% RSLogix 500 project LVD190424_LVD.RSS, saved by version 11.00.00.00 %
PROJECT "LINCEBOT"    % processor: MicroLogix 1400 %

PROGRAM FILES
  LAD 2 "MAIN"  65 rungs  % Main Program Routine %
  LAD 4 "PACKAGER"  20 rungs  % normal %
  LAD 6 "TIMING"  11 rungs  % normal %
  LAD 8 "LOOP TIME"  6 rungs
  LAD 10 "AIR PRESUR"  2 rungs
  LAD 12 "ENABLES"  14 rungs
  LAD 14 "SPEED OUT"  12 rungs
  LAD 16 "TOTALCOUNT"  4 rungs
  LAD 18 "TESTTRIG1"  3 rungs
  LAD 20 "TESTTRIG5"  3 rungs
  LAD 22 "TESTTRIG6"  3 rungs
  LAD 24 "SKIPPED"  5 rungs
  LAD 26 "TEST TIME"  11 rungs
  LAD 70 "ALIGNFAILS"  4 rungs  % normal %
  LAD 80 "HSC BOT"  5 rungs
  LAD 90 "HSC TOP"  5 rungs
  LAD 100 "1 MS STI"  24 rungs  % high speed %
  LAD 102 "SPEED BOT"  8 rungs  % high speed %
  LAD 103 "SPEED TOP"  8 rungs  % high speed %
  LAD 104 "P BOT"  9 rungs  % high speed %
  LAD 105 "P TOP"  8 rungs  % high speed %
  LAD 110 "SHIFT BOT"  9 rungs
  LAD 111 "SHIFT TOP"  13 rungs
  LAD 120 "BOTOPTIC"  3 rungs
  LAD 121 "BOTOPTMES"  7 rungs
  LAD 124 "INS1RESULT"  10 rungs
  LAD 125 "FIXERR1"  8 rungs
  LAD 127 "INS1"  40 rungs
  LAD 128 "INS1PASS"  4 rungs
  LAD 129 "INS1ACQ"  11 rungs
  LAD 130 "INS1TRIG"  9 rungs
  LAD 131 "XFER"  2 rungs
  LAD 140 "TOPOPTIC"  7 rungs
  LAD 141 "TOPOPVERT"  3 rungs
  LAD 142 "TOPOPREAL"  7 rungs
  LAD 143 "TOPOPTEST"  15 rungs
  LAD 144 "TOPOPOKAY"  6 rungs
  LAD 149 "INS5RESULT"  10 rungs
  LAD 150 "FIXERR5"  8 rungs
  LAD 152 "INS5"  35 rungs
  LAD 153 "INS5PASS"  4 rungs
  LAD 154 "INS5ACQ"  11 rungs
  LAD 155 "INS5TRIG"  9 rungs
  LAD 159 "INS6RESULT"  10 rungs
  LAD 160 "FIXERR6"  8 rungs
  LAD 162 "INS6"  29 rungs
  LAD 163 "INS6PASS"  4 rungs
  LAD 164 "INS6ACQ"  10 rungs
  LAD 165 "INS6TRIG"  9 rungs
  LAD 170 "PASS BLOW"  11 rungs
  LAD 180 "RATE"  14 rungs
  LAD 200 "TESTOPTIC"  6 rungs
  LAD 201 "UNUSED"  19 rungs
  LAD 255 "BLANK"  11 rungs

DATA FILES
  O0 OUTPUT  11 elements
  I1 INPUT  11 elements
  S2 STATUS  66 elements
  B3 BINARY  14 elements
  T4 TIMER  40 elements
  C5 COUNTER  1 elements
  R6 CONTROL  20 elements
  N7 INTEGER  200 elements
  F8 FLOAT  100 elements
  B9 TOP BS DAT  256 elements
  B10 OLD_COM  1 elements
  B11 BOT BS DAT  256 elements
  B12 HMI_BINARY  22 elements  % general use with hmi to avoid additional reads %
  L13  COUNTS  256 elements
  F14 HMI_FLOATS  100 elements
  N15 HMI_INTS  100 elements
  L16 HMI_LONGS  100 elements
  B17 SIDE DATA  128 elements
  B18 TOP DATA  128 elements
  L19 INS1TIME  10 elements
  L20 INS1POS  10 elements
  L21 INS5TIME  10 elements
  L22 INS5POS  10 elements
  L23 NEW READ  100 elements
  L24 NEW WRITE  100 elements
  L25 INS6TIME  10 elements
  L26 INS6POS  10 elements
  L42   52 elements
  B181 BLANK  256 elements  % used to wipe bs files %
  F182 TEST FLOAT  50 elements
  L183 TEST LONG  50 elements
  N184 TEST INTS  50 elements
  B185 TEST BITS  50 elements
  N186 HMI INTS  50 elements
  L187 HMI LONG  50 elements
  F188 HMI FLOAT  50 elements
  B189 HMI BITS  50 elements
  L190 COUNTS  50 elements
  B191 ERROR BITS  10 elements
  L192 SPD OFFSET  50 elements
  F193 SPD OFFSET  50 elements
  B194 BOT GOOD  128 elements
  B195 TOP GOOD  128 elements
  B196 CTRL BITS  50 elements
  N197 CTRL INTS  50 elements
  B198 TRK BITS  50 elements
  L199 TRK LONG  50 elements
  N200 TRK INTS  50 elements
  L201 INS LONG  50 elements
  B202 INS BITS  50 elements
  N203 INS INTS  50 elements
  L204 CTRL LONG  50 elements
  F205 CTRL FLTS  50 elements

LADDER 2 "MAIN"    % Main Program Routine %
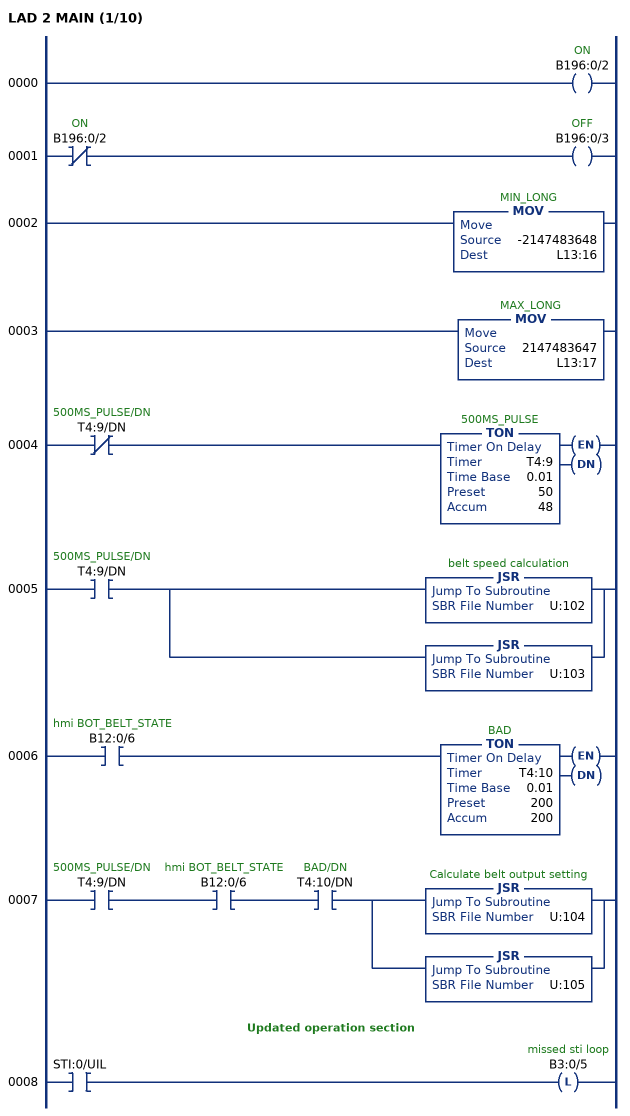
% Rung: 0 %
SOR OTE B196:0/2 EOR
%   B196:0/2  ON %
% Rung: 1 %
SOR XIO B196:0/2 OTE B196:0/3 EOR
%   B196:0/2  ON %
%   B196:0/3  OFF %
% Rung: 2 %
SOR MOV -2147483648 L13:16 EOR
%   L13:16  MIN_LONG %
% Rung: 3 %
SOR MOV 2147483647 L13:17 EOR
%   L13:17  MAX_LONG %
% Rung: 4 %
SOR XIO T4:9/DN TON T4:9 0.01 50 48 EOR
%   T4:9  500MS_PULSE %
% Rung: 5 %
SOR XIC T4:9/DN BST JSR U:102 NXB JSR U:103 BND EOR
%   T4:9  500MS_PULSE %
%   U:102  "belt speed calculation" %
% Rung: 6 %
SOR XIC B12:0/6 TON T4:10 0.01 200 200 EOR
%   B12:0/6  BOT_BELT_STATE  "hmi" %
%   T4:10  BAD %
% Rung: 7 %
SOR XIC T4:9/DN XIC B12:0/6 XIC T4:10/DN BST JSR U:104 NXB JSR U:105 BND EOR
%   T4:9  500MS_PULSE %
%   B12:0/6  BOT_BELT_STATE  "hmi" %
%   T4:10  BAD %
%   U:104  "Calculate belt output setting" %
% Rung: 8 %
% TITLE: Updated operation section %
SOR XIC STI:0/UIL OTL B3:0/5 EOR
%   B3:0/5  "missed sti loop" %

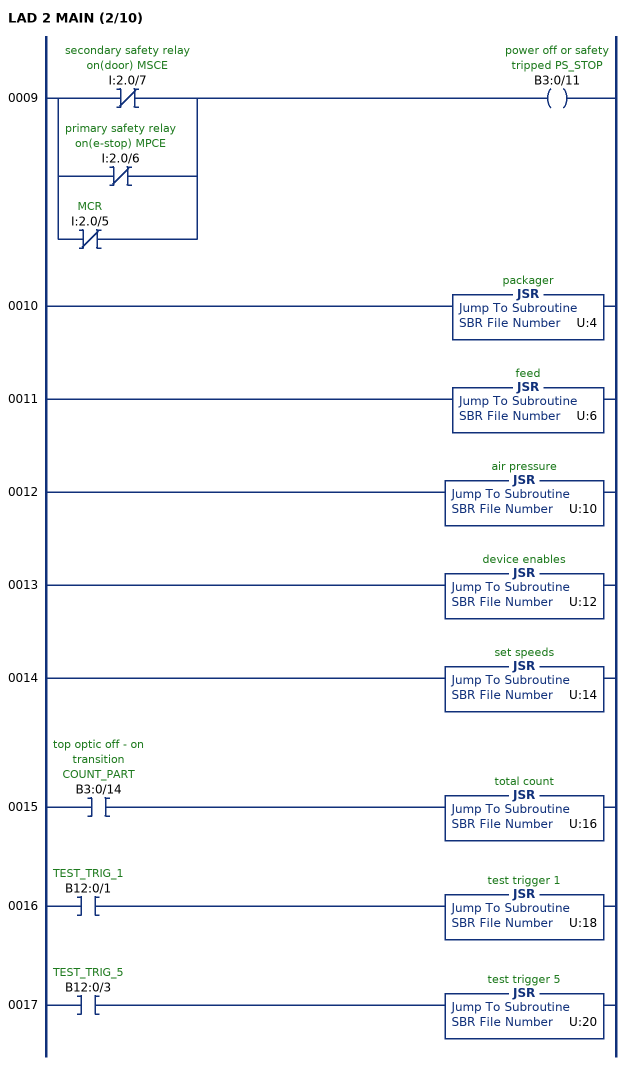
% Rung: 9 %
SOR BST XIO I:2.0/7 NXB XIO I:2.0/6 NXB XIO I:2.0/5 BND OTE B3:0/11 EOR
%   I:2.0/7  MSCE  "secondary safety relay on(door)" %
%   I:2.0/6  MPCE  "primary safety relay on(e-stop)" %
%   I:2.0/5  MCR %
%   B3:0/11  PS_STOP  "power off or safety tripped" %
% Rung: 10 %
SOR JSR U:4 EOR
%   U:4  "packager" %
% Rung: 11 %
SOR JSR U:6 EOR
%   U:6  "feed" %
% Rung: 12 %
SOR JSR U:10 EOR
%   U:10  "air pressure" %
% Rung: 13 %
SOR JSR U:12 EOR
%   U:12  "device enables" %
% Rung: 14 %
SOR JSR U:14 EOR
%   U:14  "set speeds" %
% Rung: 15 %
SOR XIC B3:0/14 JSR U:16 EOR
%   B3:0/14  COUNT_PART  "top optic off - on transition" %
%   U:16  "total count" %
% Rung: 16 %
SOR XIC B12:0/1 JSR U:18 EOR
%   B12:0/1  TEST_TRIG_1 %
%   U:18  "test trigger 1" %
% Rung: 17 %
SOR XIC B12:0/3 JSR U:20 EOR
%   B12:0/3  TEST_TRIG_5 %
%   U:20  "test trigger 5" %

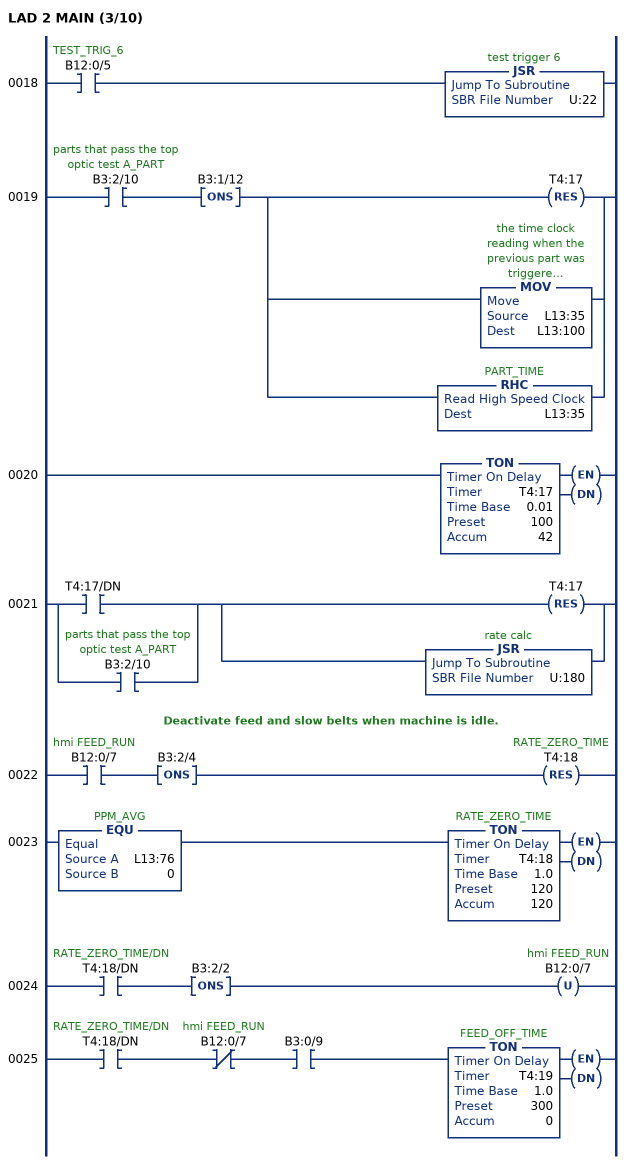
% Rung: 18 %
SOR XIC B12:0/5 JSR U:22 EOR
%   B12:0/5  TEST_TRIG_6 %
%   U:22  "test trigger 6" %
% Rung: 19 %
SOR XIC B3:2/10 ONS B3:1/12 BST RES T4:17 NXB MOV L13:35 L13:100 NXB RHC L13:35 BND EOR
%   B3:2/10  A_PART  "parts that pass the top optic test" %
%   L13:35  PART_TIME %
%   L13:100  LAST_PART_TIME  "the time clock reading when the previous part was triggered" %
% Rung: 20 %
SOR TON T4:17 0.01 100 42 EOR
% Rung: 21 %
SOR BST XIC T4:17/DN NXB XIC B3:2/10 BND BST RES T4:17 NXB JSR U:180 BND EOR
%   B3:2/10  A_PART  "parts that pass the top optic test" %
%   U:180  "rate calc" %
% Rung: 22 %
% TITLE: Deactivate feed and slow belts when machine is idle. %
SOR XIC B12:0/7 ONS B3:2/4 RES T4:18 EOR
%   B12:0/7  FEED_RUN  "hmi" %
%   T4:18  RATE_ZERO_TIME %
% Rung: 23 %
SOR EQU L13:76 0 TON T4:18 1.0 120 120 EOR
%   L13:76  PPM_AVG %
%   T4:18  RATE_ZERO_TIME %
% Rung: 24 %
SOR XIC T4:18/DN ONS B3:2/2 OTU B12:0/7 EOR
%   T4:18  RATE_ZERO_TIME %
%   B12:0/7  FEED_RUN  "hmi" %
% Rung: 25 %
SOR XIC T4:18/DN XIO B12:0/7 XIC B3:0/9 TON T4:19 1.0 300 0 EOR
%   T4:18  RATE_ZERO_TIME %
%   B12:0/7  FEED_RUN  "hmi" %
%   T4:19  FEED_OFF_TIME %

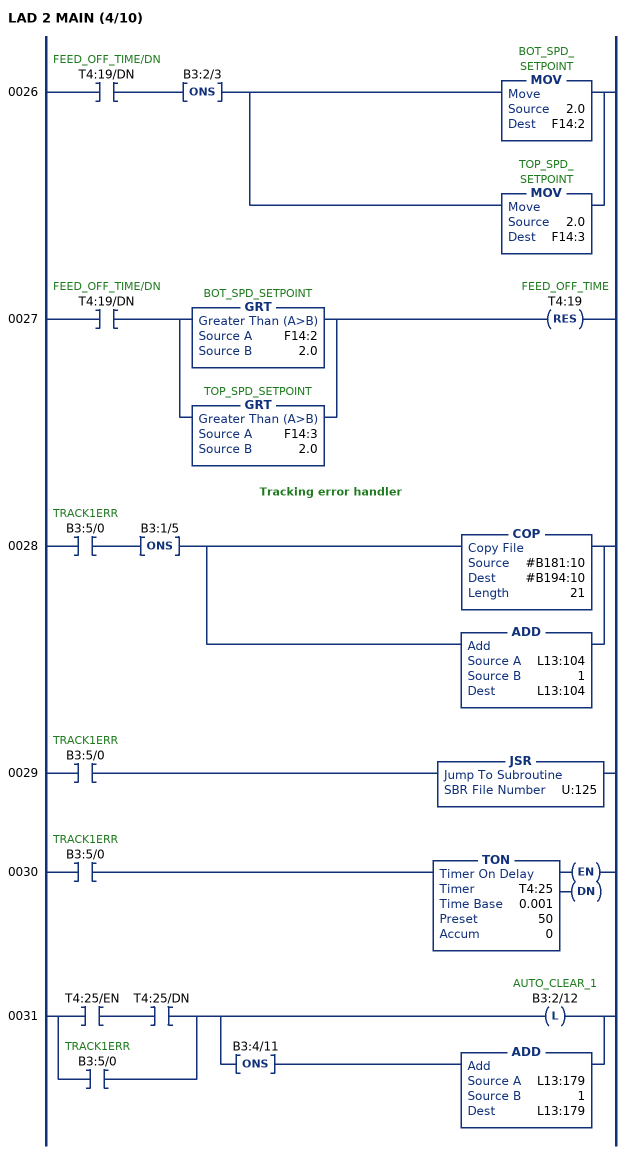
% Rung: 26 %
SOR XIC T4:19/DN ONS B3:2/3 BST MOV 2.0 F14:2 NXB MOV 2.0 F14:3 BND EOR
%   T4:19  FEED_OFF_TIME %
%   F14:2  BOT_SPD_SETPOINT %
%   F14:3  TOP_SPD_SETPOINT %
% Rung: 27 %
SOR XIC T4:19/DN BST GRT F14:2 2.0 NXB GRT F14:3 2.0 BND RES T4:19 EOR
%   T4:19  FEED_OFF_TIME %
%   F14:2  BOT_SPD_SETPOINT %
%   F14:3  TOP_SPD_SETPOINT %
% Rung: 28 %
% TITLE: Tracking error handler %
SOR XIC B3:5/0 ONS B3:1/5 BST COP #B181:10 #B194:10 21 NXB ADD L13:104 1 L13:104 BND EOR
%   B3:5/0  TRACK1ERR %
% Rung: 29 %
SOR XIC B3:5/0 JSR U:125 EOR
%   B3:5/0  TRACK1ERR %
% Rung: 30 %
SOR XIC B3:5/0 TON T4:25 0.001 50 0 EOR
%   B3:5/0  TRACK1ERR %
% Rung: 31 %
SOR BST XIC T4:25/EN XIC T4:25/DN NXB XIC B3:5/0 BND BST OTL B3:2/12 NXB ONS B3:4/11 ADD L13:179 1 L13:179 BND EOR
%   B3:5/0  TRACK1ERR %
%   B3:2/12  AUTO_CLEAR_1 %

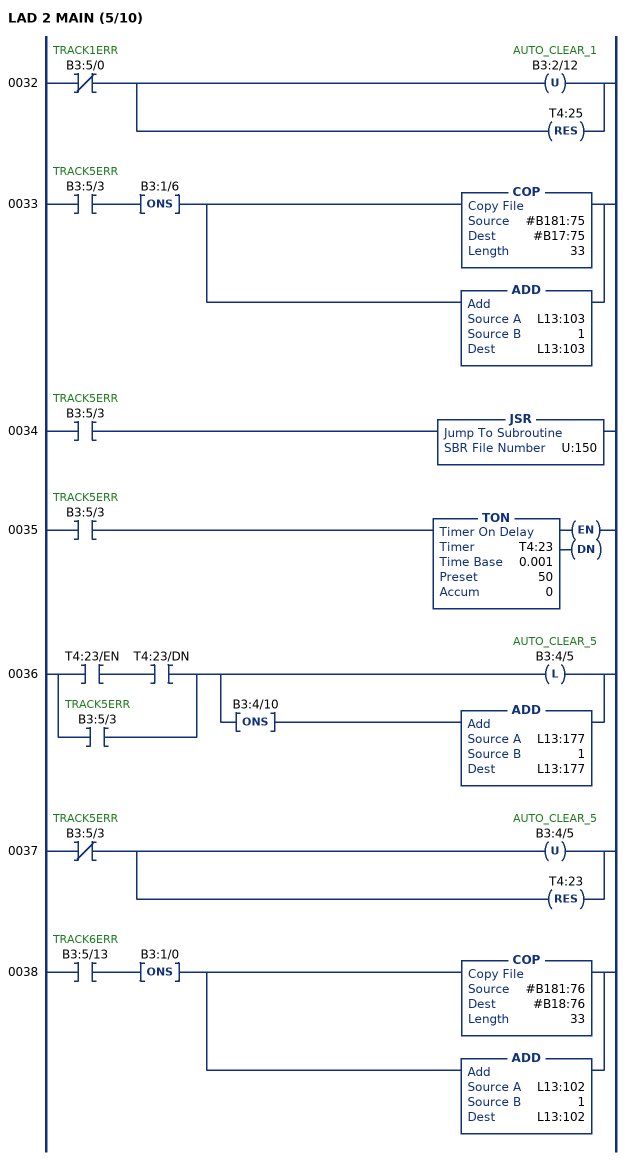
% Rung: 32 %
SOR XIO B3:5/0 BST OTU B3:2/12 NXB RES T4:25 BND EOR
%   B3:5/0  TRACK1ERR %
%   B3:2/12  AUTO_CLEAR_1 %
% Rung: 33 %
SOR XIC B3:5/3 ONS B3:1/6 BST COP #B181:75 #B17:75 33 NXB ADD L13:103 1 L13:103 BND EOR
%   B3:5/3  TRACK5ERR %
% Rung: 34 %
SOR XIC B3:5/3 JSR U:150 EOR
%   B3:5/3  TRACK5ERR %
% Rung: 35 %
SOR XIC B3:5/3 TON T4:23 0.001 50 0 EOR
%   B3:5/3  TRACK5ERR %
% Rung: 36 %
SOR BST XIC T4:23/EN XIC T4:23/DN NXB XIC B3:5/3 BND BST OTL B3:4/5 NXB ONS B3:4/10 ADD L13:177 1 L13:177 BND EOR
%   B3:5/3  TRACK5ERR %
%   B3:4/5  AUTO_CLEAR_5 %
% Rung: 37 %
SOR XIO B3:5/3 BST OTU B3:4/5 NXB RES T4:23 BND EOR
%   B3:5/3  TRACK5ERR %
%   B3:4/5  AUTO_CLEAR_5 %
% Rung: 38 %
SOR XIC B3:5/13 ONS B3:1/0 BST COP #B181:76 #B18:76 33 NXB ADD L13:102 1 L13:102 BND EOR
%   B3:5/13  TRACK6ERR %

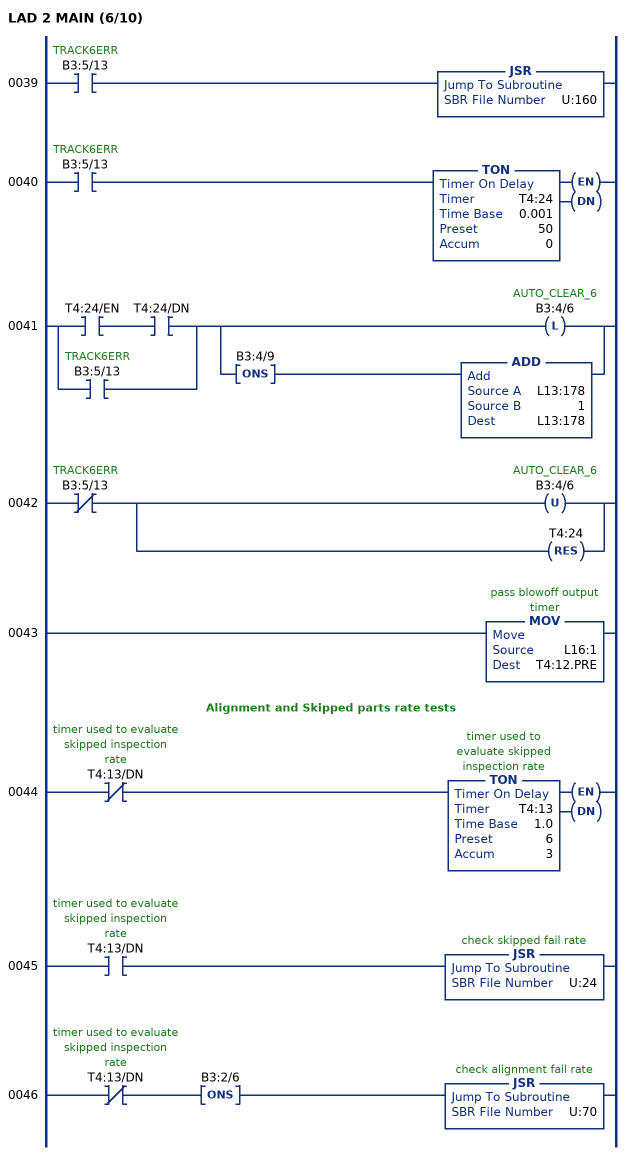
% Rung: 39 %
SOR XIC B3:5/13 JSR U:160 EOR
%   B3:5/13  TRACK6ERR %
% Rung: 40 %
SOR XIC B3:5/13 TON T4:24 0.001 50 0 EOR
%   B3:5/13  TRACK6ERR %
% Rung: 41 %
SOR BST XIC T4:24/EN XIC T4:24/DN NXB XIC B3:5/13 BND BST OTL B3:4/6 NXB ONS B3:4/9 ADD L13:178 1 L13:178 BND EOR
%   B3:5/13  TRACK6ERR %
%   B3:4/6  AUTO_CLEAR_6 %
% Rung: 42 %
SOR XIO B3:5/13 BST OTU B3:4/6 NXB RES T4:24 BND EOR
%   B3:5/13  TRACK6ERR %
%   B3:4/6  AUTO_CLEAR_6 %
% Rung: 43 %
SOR MOV L16:1 T4:12.PRE EOR
%   L16:1  BLOW_TIME %
%   T4:12  "pass blowoff output timer" %
% Rung: 44 %
% TITLE: Alignment and Skipped parts rate tests %
SOR XIO T4:13/DN TON T4:13 1.0 6 3 EOR
%   T4:13  "timer used to evaluate skipped inspection rate" %
% Rung: 45 %
SOR XIC T4:13/DN JSR U:24 EOR
%   T4:13  "timer used to evaluate skipped inspection rate" %
%   U:24  "check skipped fail rate" %
% Rung: 46 %
SOR XIO T4:13/DN ONS B3:2/6 JSR U:70 EOR
%   T4:13  "timer used to evaluate skipped inspection rate" %
%   U:70  "check alignment fail rate" %

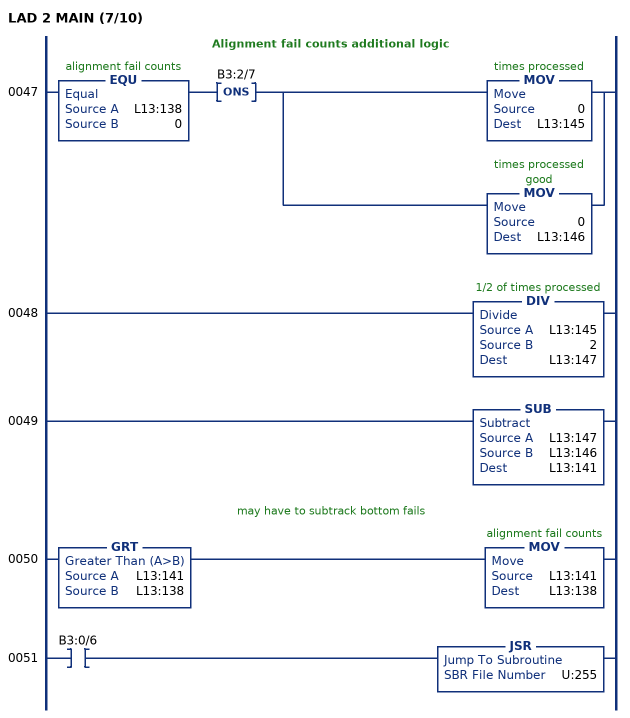
% Rung: 47 %
% TITLE: Alignment fail counts additional logic %
SOR EQU L13:138 0 ONS B3:2/7 BST MOV 0 L13:145 NXB MOV 0 L13:146 BND EOR
%   L13:138  "alignment fail counts" %
%   L13:145  "times processed" %
%   L13:146  "times processed good" %
% Rung: 48 %
SOR DIV L13:145 2 L13:147 EOR
%   L13:145  "times processed" %
%   L13:147  "1/2 of times processed" %
% Rung: 49 %
SOR SUB L13:147 L13:146 L13:141 EOR
%   L13:147  "1/2 of times processed" %
%   L13:146  "times processed good" %
% Rung: 50 %
% may have to subtrack bottom fails %
SOR GRT L13:141 L13:138 MOV L13:141 L13:138 EOR
%   L13:138  "alignment fail counts" %
% Rung: 51 %
SOR XIC B3:0/6 JSR U:255 EOR

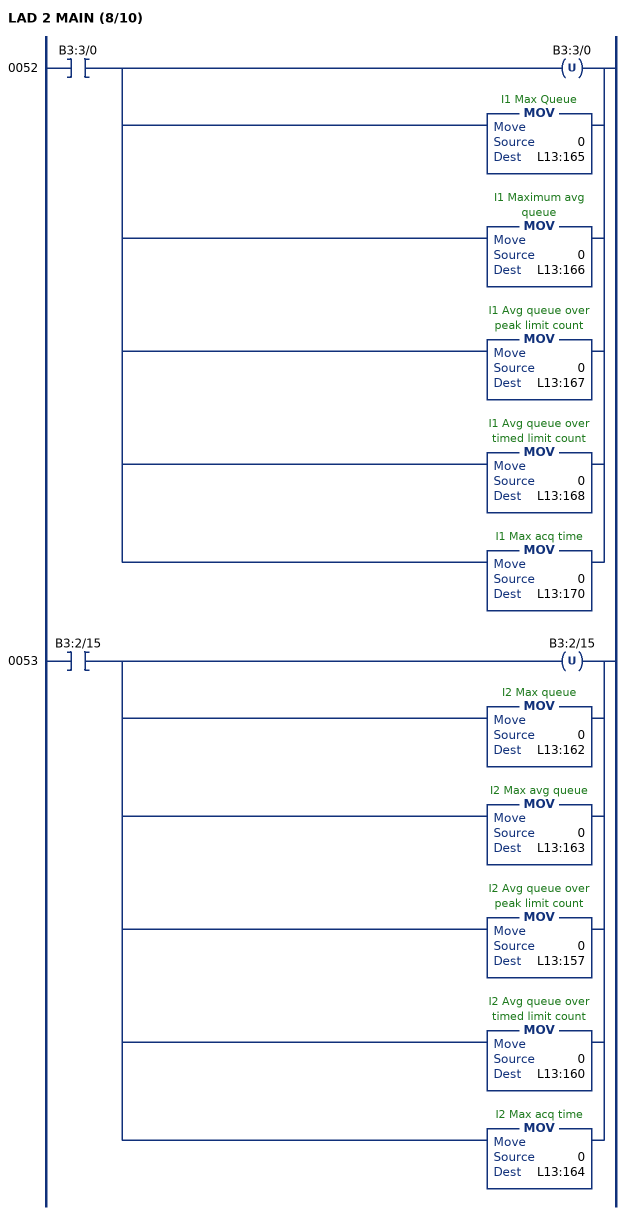
% Rung: 52 %
SOR XIC B3:3/0 BST OTU B3:3/0 NXB MOV 0 L13:165 NXB MOV 0 L13:166 NXB MOV 0 L13:167 NXB MOV 0 L13:168 NXB MOV 0 L13:170 BND EOR
%   L13:165  "I1 Max Queue" %
%   L13:166  "I1 Maximum avg queue" %
%   L13:167  "I1 Avg queue over peak limit count" %
%   L13:168  "I1 Avg queue over timed limit count" %
%   L13:170  "I1 Max acq time" %
% Rung: 53 %
SOR XIC B3:2/15 BST OTU B3:2/15 NXB MOV 0 L13:162 NXB MOV 0 L13:163 NXB MOV 0 L13:157 NXB MOV 0 L13:160 NXB MOV 0 L13:164 BND EOR
%   L13:162  "I2 Max queue" %
%   L13:163  "I2 Max avg queue" %
%   L13:157  "I2 Avg queue over peak limit count" %
%   L13:160  "I2 Avg queue over timed limit count" %
%   L13:164  "I2 Max acq time" %

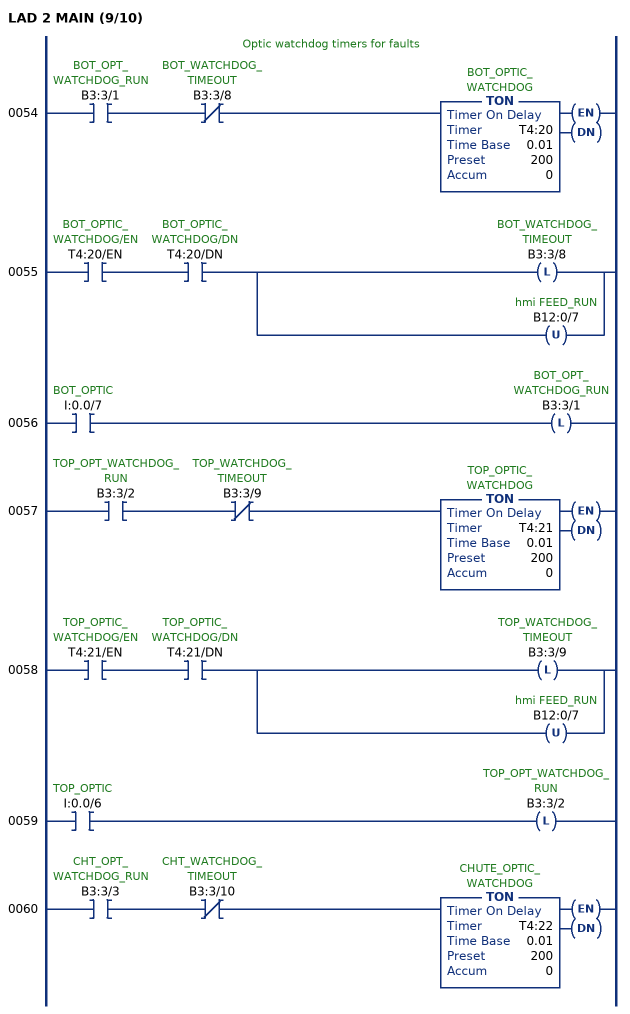
% Rung: 54 %
% Optic watchdog timers for faults %
SOR XIC B3:3/1 XIO B3:3/8 TON T4:20 0.01 200 0 EOR
%   B3:3/1  BOT_OPT_WATCHDOG_RUN %
%   B3:3/8  BOT_WATCHDOG_TIMEOUT %
%   T4:20  BOT_OPTIC_WATCHDOG %
% Rung: 55 %
SOR XIC T4:20/EN XIC T4:20/DN BST OTL B3:3/8 NXB OTU B12:0/7 BND EOR
%   T4:20  BOT_OPTIC_WATCHDOG %
%   B3:3/8  BOT_WATCHDOG_TIMEOUT %
%   B12:0/7  FEED_RUN  "hmi" %
% Rung: 56 %
SOR XIC I:0.0/7 OTL B3:3/1 EOR
%   I:0.0/7  BOT_OPTIC %
%   B3:3/1  BOT_OPT_WATCHDOG_RUN %
% Rung: 57 %
SOR XIC B3:3/2 XIO B3:3/9 TON T4:21 0.01 200 0 EOR
%   B3:3/2  TOP_OPT_WATCHDOG_RUN %
%   B3:3/9  TOP_WATCHDOG_TIMEOUT %
%   T4:21  TOP_OPTIC_WATCHDOG %
% Rung: 58 %
SOR XIC T4:21/EN XIC T4:21/DN BST OTL B3:3/9 NXB OTU B12:0/7 BND EOR
%   T4:21  TOP_OPTIC_WATCHDOG %
%   B3:3/9  TOP_WATCHDOG_TIMEOUT %
%   B12:0/7  FEED_RUN  "hmi" %
% Rung: 59 %
SOR XIC I:0.0/6 OTL B3:3/2 EOR
%   I:0.0/6  TOP_OPTIC %
%   B3:3/2  TOP_OPT_WATCHDOG_RUN %
% Rung: 60 %
SOR XIC B3:3/3 XIO B3:3/10 TON T4:22 0.01 200 0 EOR
%   B3:3/3  CHT_OPT_WATCHDOG_RUN %
%   B3:3/10  CHT_WATCHDOG_TIMEOUT %
%   T4:22  CHUTE_OPTIC_WATCHDOG %

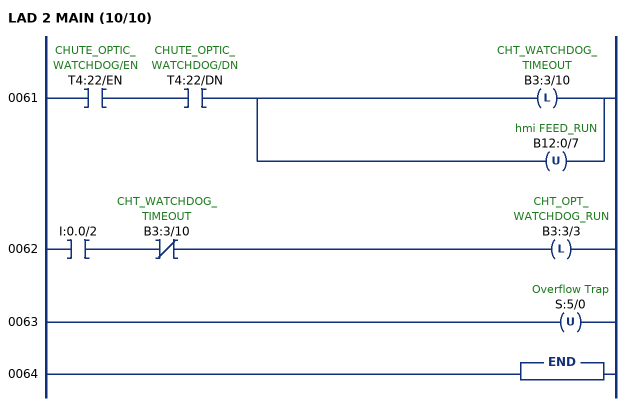
% Rung: 61 %
SOR XIC T4:22/EN XIC T4:22/DN BST OTL B3:3/10 NXB OTU B12:0/7 BND EOR
%   T4:22  CHUTE_OPTIC_WATCHDOG %
%   B3:3/10  CHT_WATCHDOG_TIMEOUT %
%   B12:0/7  FEED_RUN  "hmi" %
% Rung: 62 %
SOR XIC I:0.0/2 XIO B3:3/10 OTL B3:3/3 EOR
%   B3:3/10  CHT_WATCHDOG_TIMEOUT %
%   B3:3/3  CHT_OPT_WATCHDOG_RUN %
% Rung: 63 %
SOR OTU S:5/0 EOR
%   S:5/0  "Overflow Trap" %
% Rung: 64 %
SOR END EOR

LADDER 4 "PACKAGER"    % normal %
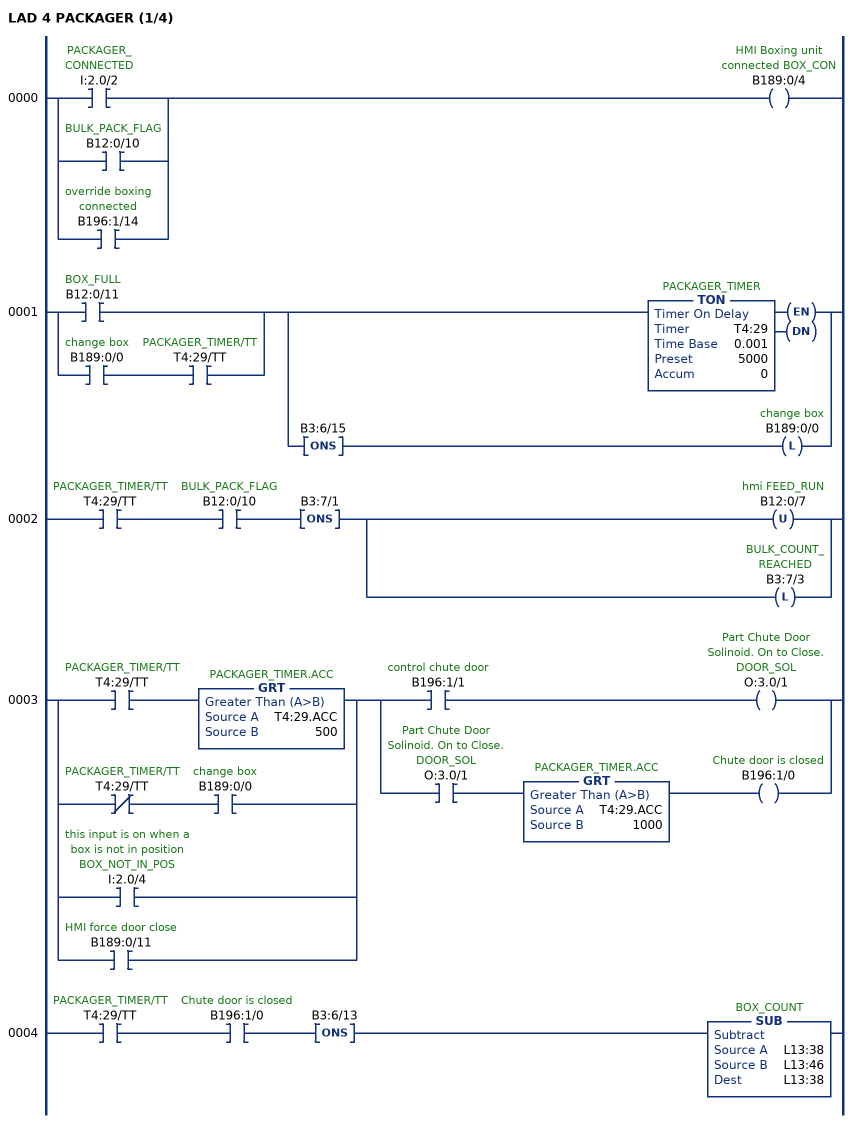
% Rung: 0 %
SOR BST XIC I:2.0/2 NXB XIC B12:0/10 NXB XIC B196:1/14 BND OTE B189:0/4 EOR
%   I:2.0/2  PACKAGER_CONNECTED %
%   B12:0/10  BULK_PACK_FLAG %
%   B196:1/14  "override boxing connected" %
%   B189:0/4  BOX_CON  "HMI Boxing unit connected" %
% Rung: 1 %
SOR BST XIC B12:0/11 NXB XIC B189:0/0 XIC T4:29/TT BND BST TON T4:29 0.001 5000 0 NXB ONS B3:6/15 OTL B189:0/0 BND EOR
%   B12:0/11  BOX_FULL %
%   B189:0/0  "change box" %
%   T4:29  PACKAGER_TIMER %
% Rung: 2 %
SOR XIC T4:29/TT XIC B12:0/10 ONS B3:7/1 BST OTU B12:0/7 NXB OTL B3:7/3 BND EOR
%   T4:29  PACKAGER_TIMER %
%   B12:0/10  BULK_PACK_FLAG %
%   B12:0/7  FEED_RUN  "hmi" %
%   B3:7/3  BULK_COUNT_REACHED %
% Rung: 3 %
SOR BST XIC T4:29/TT GRT T4:29.ACC 500 NXB XIO T4:29/TT XIC B189:0/0 NXB XIC I:2.0/4 NXB XIC B189:0/11 BND BST XIC B196:1/1 OTE O:3.0/1 NXB XIC O:3.0/1 GRT T4:29.ACC 1000 OTE B196:1/0 BND EOR
%   T4:29  PACKAGER_TIMER %
%   B189:0/0  "change box" %
%   I:2.0/4  BOX_NOT_IN_POS  "this input is on when a box is not in position" %
%   B189:0/11  "HMI force door close" %
%   B196:1/1  "control chute door" %
%   O:3.0/1  DOOR_SOL  "Part Chute Door Solinoid. On to Close." %
%   B196:1/0  "Chute door is closed" %
% Rung: 4 %
SOR XIC T4:29/TT XIC B196:1/0 ONS B3:6/13 SUB L13:38 L13:46 L13:38 EOR
%   T4:29  PACKAGER_TIMER %
%   B196:1/0  "Chute door is closed" %
%   L13:38  BOX_COUNT %
%   L13:46  BOX_LIMIT  "box count setpoint" %

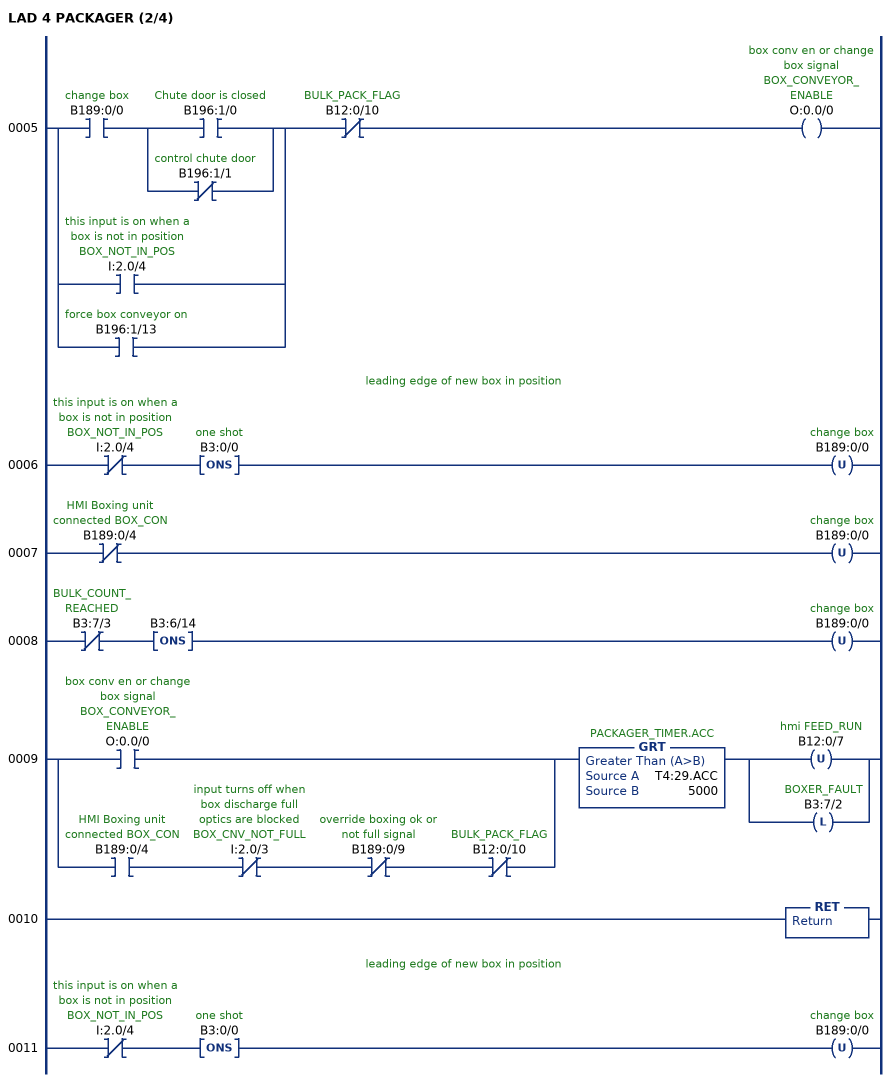
% Rung: 5 %
SOR BST XIC B189:0/0 BST XIC B196:1/0 NXB XIO B196:1/1 BND NXB XIC I:2.0/4 NXB XIC B196:1/13 BND XIO B12:0/10 OTE O:0.0/0 EOR
%   B189:0/0  "change box" %
%   B196:1/0  "Chute door is closed" %
%   B196:1/1  "control chute door" %
%   I:2.0/4  BOX_NOT_IN_POS  "this input is on when a box is not in position" %
%   B196:1/13  "force box conveyor on" %
%   B12:0/10  BULK_PACK_FLAG %
%   O:0.0/0  BOX_CONVEYOR_ENABLE  "box conv en or change box signal" %
% Rung: 6 %
% leading edge of new box in position %
SOR XIO I:2.0/4 ONS B3:0/0 OTU B189:0/0 EOR
%   I:2.0/4  BOX_NOT_IN_POS  "this input is on when a box is not in position" %
%   B3:0/0  "one shot" %
%   B189:0/0  "change box" %
% Rung: 7 %
SOR XIO B189:0/4 OTU B189:0/0 EOR
%   B189:0/4  BOX_CON  "HMI Boxing unit connected" %
%   B189:0/0  "change box" %
% Rung: 8 %
SOR XIO B3:7/3 ONS B3:6/14 OTU B189:0/0 EOR
%   B3:7/3  BULK_COUNT_REACHED %
%   B189:0/0  "change box" %
% Rung: 9 %
SOR BST XIC O:0.0/0 NXB XIC B189:0/4 XIO I:2.0/3 XIO B189:0/9 XIO B12:0/10 BND GRT T4:29.ACC 5000 BST OTU B12:0/7 NXB OTL B3:7/2 BND EOR
%   O:0.0/0  BOX_CONVEYOR_ENABLE  "box conv en or change box signal" %
%   B189:0/4  BOX_CON  "HMI Boxing unit connected" %
%   I:2.0/3  BOX_CNV_NOT_FULL  "input turns off when box discharge full optics are blocked" %
%   B189:0/9  "override boxing ok or not full signal" %
%   B12:0/10  BULK_PACK_FLAG %
%   T4:29  PACKAGER_TIMER %
%   B12:0/7  FEED_RUN  "hmi" %
%   B3:7/2  BOXER_FAULT %
% Rung: 10 %
SOR RET EOR
% Rung: 11 %
% leading edge of new box in position %
SOR XIO I:2.0/4 ONS B3:0/0 OTU B189:0/0 EOR
%   I:2.0/4  BOX_NOT_IN_POS  "this input is on when a box is not in position" %
%   B3:0/0  "one shot" %
%   B189:0/0  "change box" %

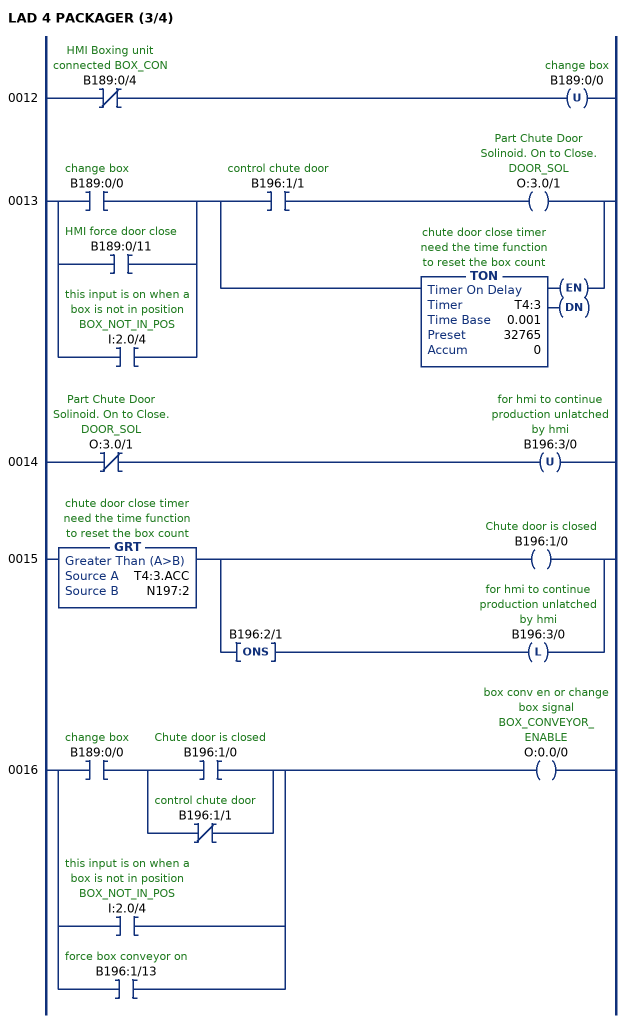
% Rung: 12 %
SOR XIO B189:0/4 OTU B189:0/0 EOR
%   B189:0/4  BOX_CON  "HMI Boxing unit connected" %
%   B189:0/0  "change box" %
% Rung: 13 %
SOR BST XIC B189:0/0 NXB XIC B189:0/11 NXB XIC I:2.0/4 BND BST XIC B196:1/1 OTE O:3.0/1 NXB TON T4:3 0.001 32765 0 BND EOR
%   B189:0/0  "change box" %
%   B189:0/11  "HMI force door close" %
%   I:2.0/4  BOX_NOT_IN_POS  "this input is on when a box is not in position" %
%   B196:1/1  "control chute door" %
%   O:3.0/1  DOOR_SOL  "Part Chute Door Solinoid. On to Close." %
%   T4:3  "chute door close timer need the time function to reset the box count" %
% Rung: 14 %
SOR XIO O:3.0/1 OTU B196:3/0 EOR
%   O:3.0/1  DOOR_SOL  "Part Chute Door Solinoid. On to Close." %
%   B196:3/0  "for hmi to continue production unlatched by hmi" %
% Rung: 15 %
SOR GRT T4:3.ACC N197:2 BST OTE B196:1/0 NXB ONS B196:2/1 OTL B196:3/0 BND EOR
%   T4:3  "chute door close timer need the time function to reset the box count" %
%   N197:2  "time for chute door to close" %
%   B196:1/0  "Chute door is closed" %
%   B196:3/0  "for hmi to continue production unlatched by hmi" %
% Rung: 16 %
SOR BST XIC B189:0/0 BST XIC B196:1/0 NXB XIO B196:1/1 BND NXB XIC I:2.0/4 NXB XIC B196:1/13 BND OTE O:0.0/0 EOR
%   B189:0/0  "change box" %
%   B196:1/0  "Chute door is closed" %
%   B196:1/1  "control chute door" %
%   I:2.0/4  BOX_NOT_IN_POS  "this input is on when a box is not in position" %
%   B196:1/13  "force box conveyor on" %
%   O:0.0/0  BOX_CONVEYOR_ENABLE  "box conv en or change box signal" %

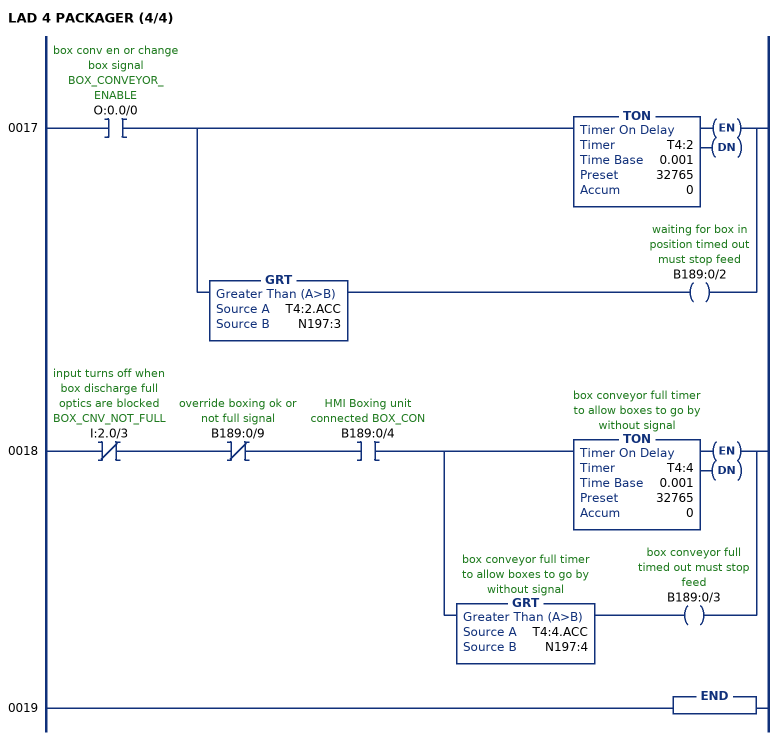
% Rung: 17 %
SOR XIC O:0.0/0 BST TON T4:2 0.001 32765 0 NXB GRT T4:2.ACC N197:3 OTE B189:0/2 BND EOR
%   O:0.0/0  BOX_CONVEYOR_ENABLE  "box conv en or change box signal" %
%   N197:3  "FeedWheel Speed Output Setting" %
%   B189:0/2  "waiting for box in position timed out must stop feed" %
% Rung: 18 %
SOR XIO I:2.0/3 XIO B189:0/9 XIC B189:0/4 BST TON T4:4 0.001 32765 0 NXB GRT T4:4.ACC N197:4 OTE B189:0/3 BND EOR
%   I:2.0/3  BOX_CNV_NOT_FULL  "input turns off when box discharge full optics are blocked" %
%   B189:0/9  "override boxing ok or not full signal" %
%   B189:0/4  BOX_CON  "HMI Boxing unit connected" %
%   T4:4  "box conveyor full timer to allow boxes to go by without signal" %
%   N197:4  "boxing convery full time out time (ms)" %
%   B189:0/3  "box conveyor full timed out must stop feed" %
% Rung: 19 %
SOR END EOR

LADDER 6 "TIMING"    % normal %
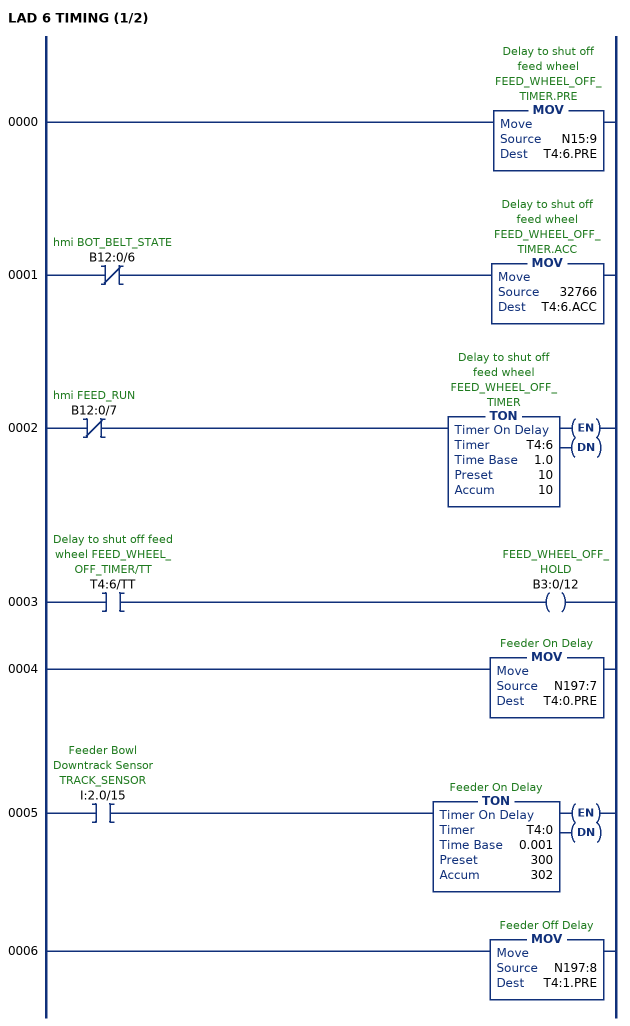
% Rung: 0 %
SOR MOV N15:9 T4:6.PRE EOR
%   N15:9  FEED_WHEEL_STOP_TIME %
%   T4:6  FEED_WHEEL_OFF_TIMER  "Delay to shut off feed wheel" %
% Rung: 1 %
SOR XIO B12:0/6 MOV 32766 T4:6.ACC EOR
%   B12:0/6  BOT_BELT_STATE  "hmi" %
%   T4:6  FEED_WHEEL_OFF_TIMER  "Delay to shut off feed wheel" %
% Rung: 2 %
SOR XIO B12:0/7 TON T4:6 1.0 10 10 EOR
%   B12:0/7  FEED_RUN  "hmi" %
%   T4:6  FEED_WHEEL_OFF_TIMER  "Delay to shut off feed wheel" %
% Rung: 3 %
SOR XIC T4:6/TT OTE B3:0/12 EOR
%   T4:6  FEED_WHEEL_OFF_TIMER  "Delay to shut off feed wheel" %
%   B3:0/12  FEED_WHEEL_OFF_HOLD %
% Rung: 4 %
SOR MOV N197:7 T4:0.PRE EOR
%   N197:7  "down track on delay" %
%   T4:0  "Feeder On Delay" %
% Rung: 5 %
SOR XIC I:2.0/15 TON T4:0 0.001 300 302 EOR
%   I:2.0/15  TRACK_SENSOR  "Feeder Bowl Downtrack Sensor" %
%   T4:0  "Feeder On Delay" %
% Rung: 6 %
SOR MOV N197:8 T4:1.PRE EOR
%   N197:8  "down track off delay" %
%   T4:1  "Feeder Off Delay" %

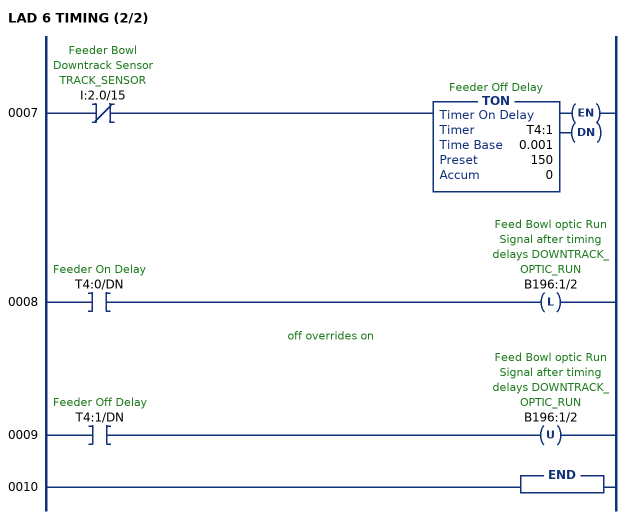
% Rung: 7 %
SOR XIO I:2.0/15 TON T4:1 0.001 150 0 EOR
%   I:2.0/15  TRACK_SENSOR  "Feeder Bowl Downtrack Sensor" %
%   T4:1  "Feeder Off Delay" %
% Rung: 8 %
SOR XIC T4:0/DN OTL B196:1/2 EOR
%   T4:0  "Feeder On Delay" %
%   B196:1/2  DOWNTRACK_OPTIC_RUN  "Feed Bowl optic Run Signal after timing delays" %
% Rung: 9 %
% off overrides on %
SOR XIC T4:1/DN OTU B196:1/2 EOR
%   T4:1  "Feeder Off Delay" %
%   B196:1/2  DOWNTRACK_OPTIC_RUN  "Feed Bowl optic Run Signal after timing delays" %
% Rung: 10 %
SOR END EOR

LADDER 8 "LOOP TIME"
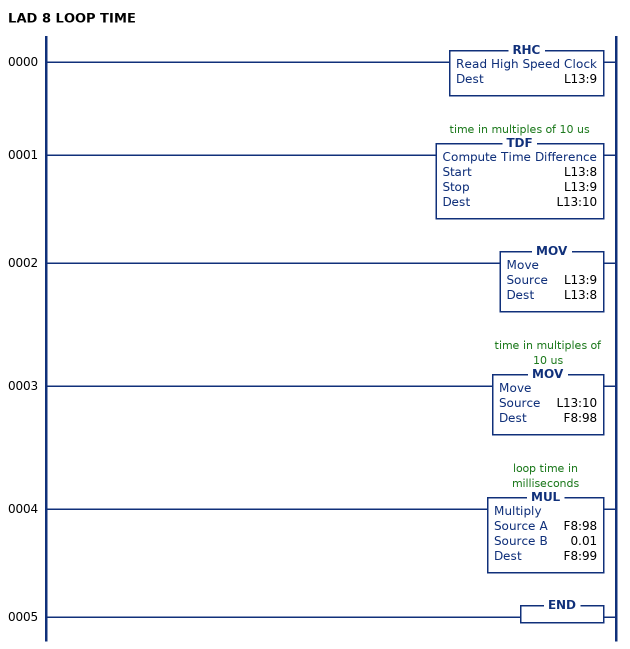
% Rung: 0 %
SOR RHC L13:9 EOR
% Rung: 1 %
SOR TDF L13:8 L13:9 L13:10 EOR
%   L13:10  "time in multiples of 10 us" %
% Rung: 2 %
SOR MOV L13:9 L13:8 EOR
% Rung: 3 %
SOR MOV L13:10 F8:98 EOR
%   L13:10  "time in multiples of 10 us" %
%   F8:98  "time in multiples of 10 us" %
% Rung: 4 %
SOR MUL F8:98 0.01 F8:99 EOR
%   F8:98  "time in multiples of 10 us" %
%   F8:99  "loop time in milliseconds" %
% Rung: 5 %
SOR END EOR

LADDER 10 "AIR PRESUR"
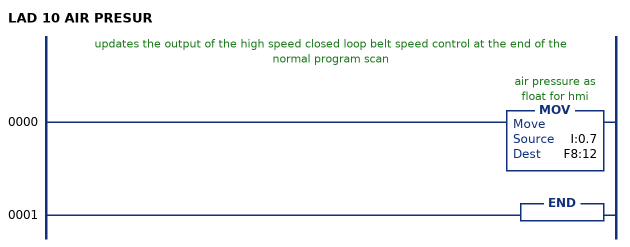
% Rung: 0 %
% updates the output of the high speed closed loop belt speed control at the end of the normal program scan %
SOR MOV I:0.7 F8:12 EOR
%   I:0.7  "Air Presure Sensor Input Signal" %
%   F8:12  "air pressure as float for hmi" %
% Rung: 1 %
SOR END EOR

LADDER 12 "ENABLES"
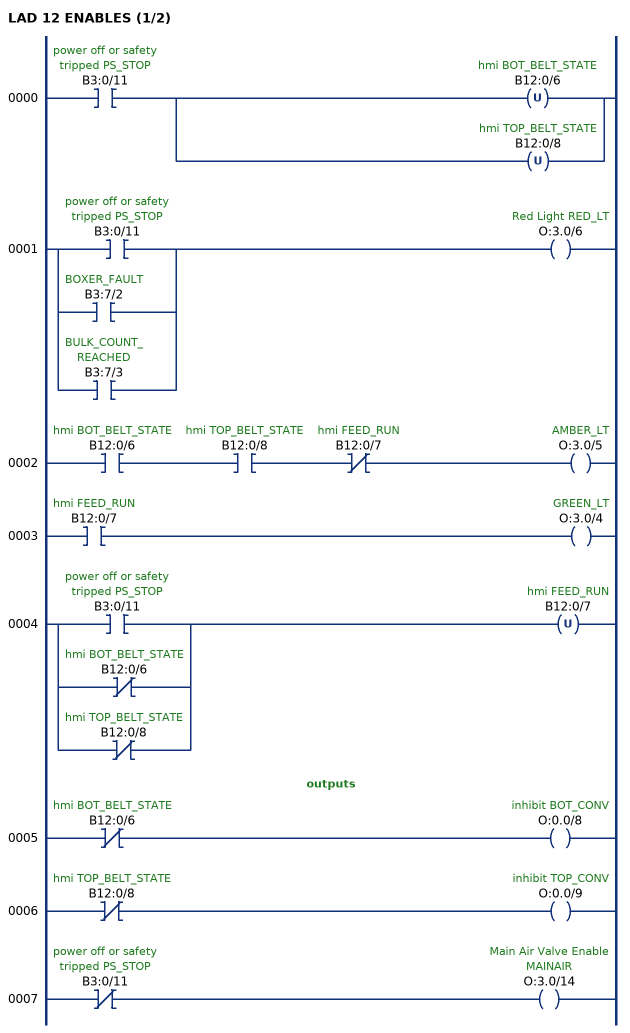
% Rung: 0 %
SOR XIC B3:0/11 BST OTU B12:0/6 NXB OTU B12:0/8 BND EOR
%   B3:0/11  PS_STOP  "power off or safety tripped" %
%   B12:0/6  BOT_BELT_STATE  "hmi" %
%   B12:0/8  TOP_BELT_STATE  "hmi" %
% Rung: 1 %
SOR BST XIC B3:0/11 NXB XIC B3:7/2 NXB XIC B3:7/3 BND OTE O:3.0/6 EOR
%   B3:0/11  PS_STOP  "power off or safety tripped" %
%   B3:7/2  BOXER_FAULT %
%   B3:7/3  BULK_COUNT_REACHED %
%   O:3.0/6  RED_LT  "Red Light" %
% Rung: 2 %
SOR XIC B12:0/6 XIC B12:0/8 XIO B12:0/7 OTE O:3.0/5 EOR
%   B12:0/6  BOT_BELT_STATE  "hmi" %
%   B12:0/8  TOP_BELT_STATE  "hmi" %
%   B12:0/7  FEED_RUN  "hmi" %
%   O:3.0/5  AMBER_LT %
% Rung: 3 %
SOR XIC B12:0/7 OTE O:3.0/4 EOR
%   B12:0/7  FEED_RUN  "hmi" %
%   O:3.0/4  GREEN_LT %
% Rung: 4 %
SOR BST XIC B3:0/11 NXB XIO B12:0/6 NXB XIO B12:0/8 BND OTU B12:0/7 EOR
%   B3:0/11  PS_STOP  "power off or safety tripped" %
%   B12:0/6  BOT_BELT_STATE  "hmi" %
%   B12:0/8  TOP_BELT_STATE  "hmi" %
%   B12:0/7  FEED_RUN  "hmi" %
% Rung: 5 %
% TITLE: outputs %
SOR XIO B12:0/6 OTE O:0.0/8 EOR
%   B12:0/6  BOT_BELT_STATE  "hmi" %
%   O:0.0/8  BOT_CONV  "inhibit" %
% Rung: 6 %
SOR XIO B12:0/8 OTE O:0.0/9 EOR
%   B12:0/8  TOP_BELT_STATE  "hmi" %
%   O:0.0/9  TOP_CONV  "inhibit" %
% Rung: 7 %
SOR XIO B3:0/11 OTE O:3.0/14 EOR
%   B3:0/11  PS_STOP  "power off or safety tripped" %
%   O:3.0/14  MAINAIR  "Main Air Valve Enable" %

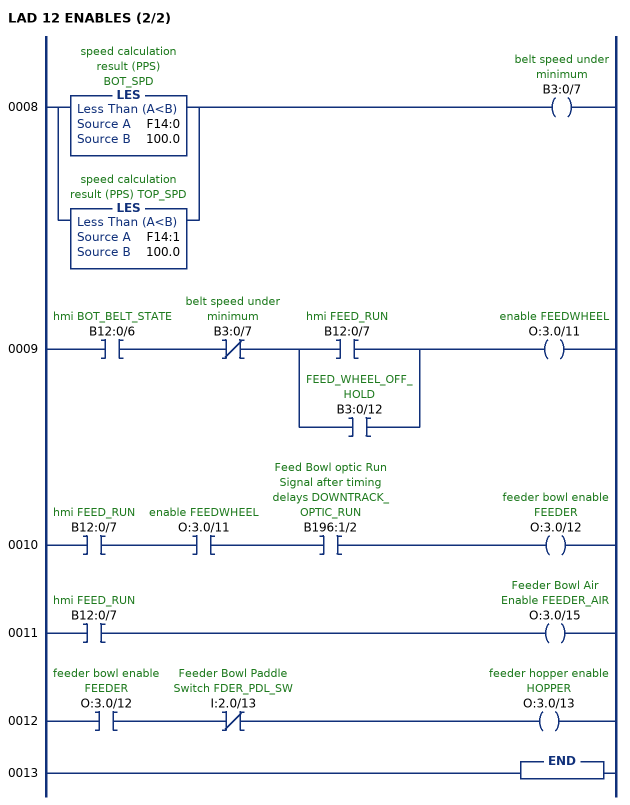
% Rung: 8 %
SOR BST LES F14:0 100.0 NXB LES F14:1 100.0 BND OTE B3:0/7 EOR
%   F14:0  BOT_SPD  "speed calculation result (PPS)" %
%   F14:1  TOP_SPD  "speed calculation result (PPS)" %
%   B3:0/7  "belt speed under minimum" %
% Rung: 9 %
SOR XIC B12:0/6 XIO B3:0/7 BST XIC B12:0/7 NXB XIC B3:0/12 BND OTE O:3.0/11 EOR
%   B12:0/6  BOT_BELT_STATE  "hmi" %
%   B3:0/7  "belt speed under minimum" %
%   B12:0/7  FEED_RUN  "hmi" %
%   B3:0/12  FEED_WHEEL_OFF_HOLD %
%   O:3.0/11  FEEDWHEEL  "enable" %
% Rung: 10 %
SOR XIC B12:0/7 XIC O:3.0/11 XIC B196:1/2 OTE O:3.0/12 EOR
%   B12:0/7  FEED_RUN  "hmi" %
%   O:3.0/11  FEEDWHEEL  "enable" %
%   B196:1/2  DOWNTRACK_OPTIC_RUN  "Feed Bowl optic Run Signal after timing delays" %
%   O:3.0/12  FEEDER  "feeder bowl enable" %
% Rung: 11 %
SOR XIC B12:0/7 OTE O:3.0/15 EOR
%   B12:0/7  FEED_RUN  "hmi" %
%   O:3.0/15  FEEDER_AIR  "Feeder Bowl Air Enable" %
% Rung: 12 %
SOR XIC O:3.0/12 XIO I:2.0/13 OTE O:3.0/13 EOR
%   O:3.0/12  FEEDER  "feeder bowl enable" %
%   I:2.0/13  FDER_PDL_SW  "Feeder Bowl Paddle Switch" %
%   O:3.0/13  HOPPER  "feeder hopper enable" %
% Rung: 13 %
SOR END EOR

LADDER 14 "SPEED OUT"
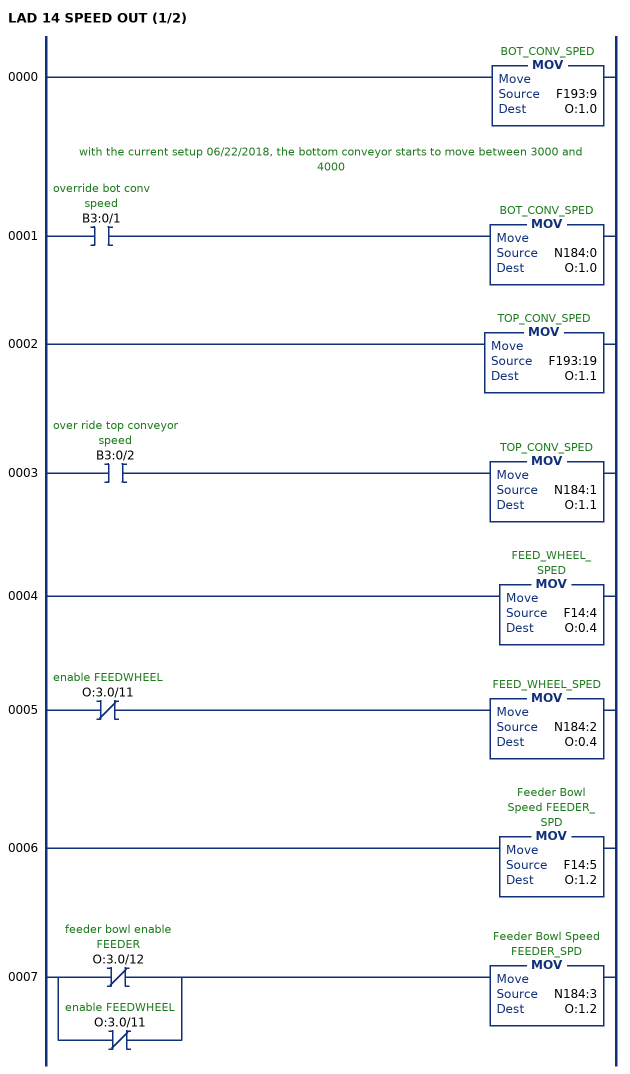
% Rung: 0 %
SOR MOV F193:9 O:1.0 EOR
%   F193:9  SCALED_BOT_VALUE %
%   O:1.0  BOT_CONV_SPED %
% Rung: 1 %
% with the current setup 06/22/2018, the bottom conveyor starts to move between 3000 and 4000 %
SOR XIC B3:0/1 MOV N184:0 O:1.0 EOR
%   B3:0/1  "override bot conv speed" %
%   O:1.0  BOT_CONV_SPED %
% Rung: 2 %
SOR MOV F193:19 O:1.1 EOR
%   F193:19  SCALED_TOP_VALUE %
%   O:1.1  TOP_CONV_SPED %
% Rung: 3 %
SOR XIC B3:0/2 MOV N184:1 O:1.1 EOR
%   B3:0/2  "over ride top conveyor speed" %
%   O:1.1  TOP_CONV_SPED %
% Rung: 4 %
SOR MOV F14:4 O:0.4 EOR
%   O:0.4  FEED_WHEEL_SPED %
% Rung: 5 %
SOR XIO O:3.0/11 MOV N184:2 O:0.4 EOR
%   O:3.0/11  FEEDWHEEL  "enable" %
%   O:0.4  FEED_WHEEL_SPED %
% Rung: 6 %
SOR MOV F14:5 O:1.2 EOR
%   O:1.2  FEEDER_SPD  "Feeder Bowl Speed" %
% Rung: 7 %
SOR BST XIO O:3.0/12 NXB XIO O:3.0/11 BND MOV N184:3 O:1.2 EOR
%   O:3.0/12  FEEDER  "feeder bowl enable" %
%   O:3.0/11  FEEDWHEEL  "enable" %
%   O:1.2  FEEDER_SPD  "Feeder Bowl Speed" %

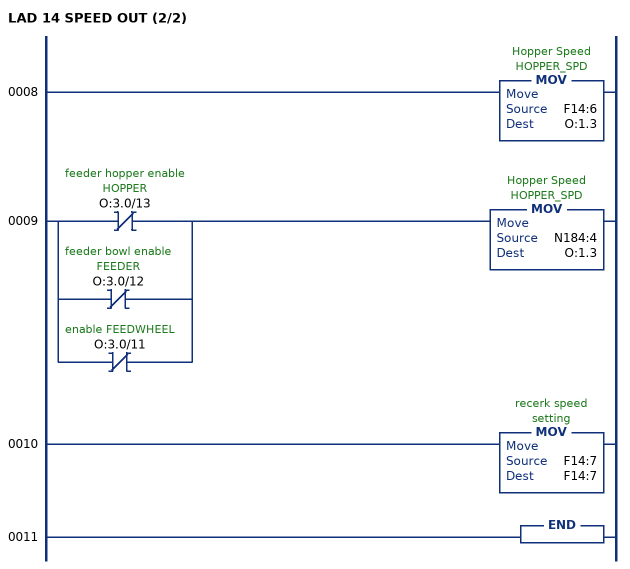
% Rung: 8 %
SOR MOV F14:6 O:1.3 EOR
%   O:1.3  HOPPER_SPD  "Hopper Speed" %
% Rung: 9 %
SOR BST XIO O:3.0/13 NXB XIO O:3.0/12 NXB XIO O:3.0/11 BND MOV N184:4 O:1.3 EOR
%   O:3.0/13  HOPPER  "feeder hopper enable" %
%   O:3.0/12  FEEDER  "feeder bowl enable" %
%   O:3.0/11  FEEDWHEEL  "enable" %
%   O:1.3  HOPPER_SPD  "Hopper Speed" %
% Rung: 10 %
SOR MOV F14:7 F14:7 EOR
%   F14:7  "recerk speed setting" %
% Rung: 11 %
SOR END EOR

LADDER 16 "TOTALCOUNT"
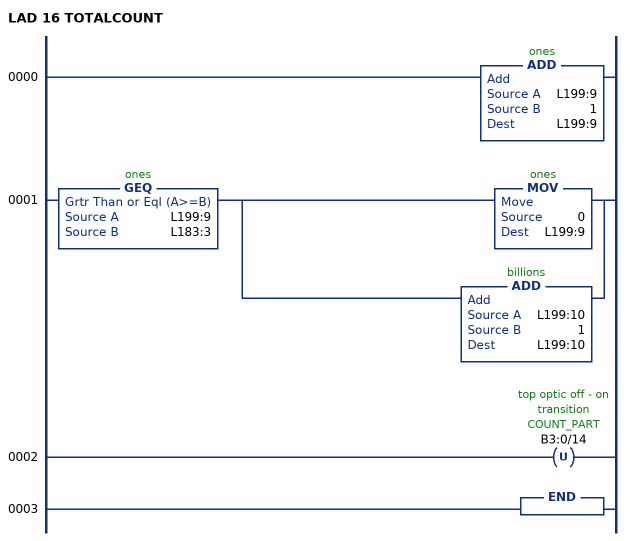
% Rung: 0 %
SOR ADD L199:9 1 L199:9 EOR
%   L199:9  "ones" %
% Rung: 1 %
SOR GEQ L199:9 L183:3 BST MOV 0 L199:9 NXB ADD L199:10 1 L199:10 BND EOR
%   L199:9  "ones" %
%   L183:3  "button state" %
%   L199:10  "billions" %
% Rung: 2 %
SOR OTU B3:0/14 EOR
%   B3:0/14  COUNT_PART  "top optic off - on transition" %
% Rung: 3 %
SOR END EOR

LADDER 18 "TESTTRIG1"
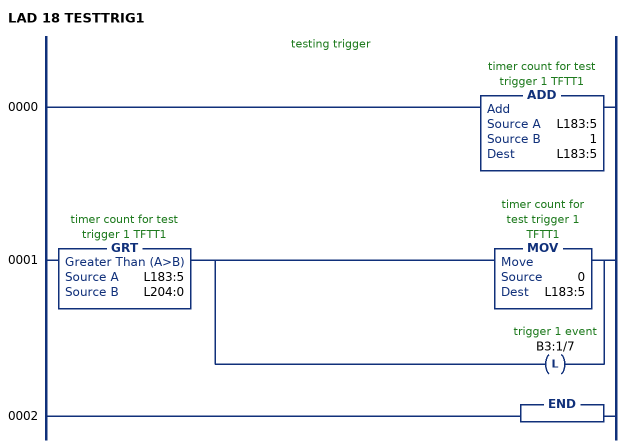
% Rung: 0 %
% testing trigger %
SOR ADD L183:5 1 L183:5 EOR
%   L183:5  TFTT1  "timer count for test trigger 1" %
% Rung: 1 %
SOR GRT L183:5 L204:0 BST MOV 0 L183:5 NXB OTL B3:1/7 BND EOR
%   L183:5  TFTT1  "timer count for test trigger 1" %
%   B3:1/7  "trigger 1 event" %
% Rung: 2 %
SOR END EOR

LADDER 20 "TESTTRIG5"
